// TIA Portal V19 export
VAR_GLOBAL   // PLC tag table "Prod_HMI_CONST"
END_VAR
VAR_GLOBAL CONSTANT   // user constants
   HMI_COLOR_LIGHT_GREY : Int := 0;
   HMI_COLOR_DARK_GREY : Int := 1;
   HMI_COLOR_RED : Int := 2;
   HMI_COLOR_GREEN : Int := 3;
END_VAR
